FUNCTION_BLOCK FB_HYST (* Basic Function Block Type *)
  (* Standard: 61499-2 *)
  (* Version 0.0, 2011-08-31, 4DIAC-IDE, 4DIAC-Consortium *)
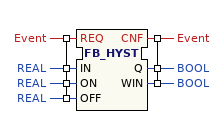
  EVENT_INPUT
    REQ WITH IN, ON, OFF; (* Normal Execution Request *)
  END_EVENT
  EVENT_OUTPUT
    CNF WITH WIN, Q; (* Execution Confirmation *)
  END_EVENT
  VAR_INPUT
    IN : REAL; (* input value *)
    ON : REAL; (* upper threshold *)
    OFF : REAL; (* lower threshold *)
  END_VAR
  VAR_OUTPUT
    Q : BOOL; (* output *)
    WIN : BOOL; (* shows that IN lies in between ON and OFF *)
  END_VAR
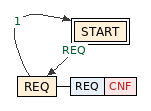
  EC_STATES
    START; (* Initial State *)
    REQ : REQ -> CNF; (* Normal execution *)
  END_STATES
  EC_TRANSITIONS
    START TO REQ := REQ;
    REQ TO START := 1;
  END_TRANSITIONS
  ALGORITHM REQ IN ST: (* Normally executed algorithm *)
IF ON >= OFF THEN
	IF IN < OFF THEN
		Q := FALSE;
		WIN := FALSE;
	ELSIF  IN > ON THEN
		Q := TRUE;
		WIN := FALSE;
	ELSE
		WIN := TRUE;
	END_IF;
ELSE
	IF IN > OFF THEN
		Q := FALSE;
		WIN := FALSE;
	ELSIF  IN < ON THEN
		Q := TRUE;
		WIN := FALSE;
	ELSE
		WIN := TRUE;
	END_IF;
END_IF;
  END_ALGORITHM
END_FUNCTION_BLOCK
